{attribute 'qualified_only' := ''}
{attribute 'strict' := ''}
TYPE cTraySize :
(
	NoSize := 0,
	Small := 1,
	Large := 2
) DINT;
END_TYPE

(* stored: Version 1.1.0.1, ProductVersion 3.1.4024.6
   DUT cTraySize: Id {9f200e47-1425-4632-b854-c8ef6bfdd896} *)
